{attribute 'pack_mode' := '1'}
TYPE ST_AnalogInputStatus_Generic :
	STRUCT
		Underrrange : BIT;
		Overrange	: BIT;
		Error		: BIT;
		WcState		: BIT;
	END_STRUCT
END_TYPE

(* stored: Version 1.1.0.1, ProductVersion 3.1.4026.18
   DUT ST_AnalogInputStatus_Generic: Id {8873af55-8532-4798-9df2-67443d859450} *)
